INTERFACE I_ChainController

METHOD addChain : I_ChainController 
VAR_INPUT
	itfChain : I_Chain;
END_VAR
END_METHOD

METHOD releaseForChain : I_ChainController
VAR_INPUT
	sChainToRelease : STRING;
	itfCommissioner : I_Chain;
END_VAR
END_METHOD

METHOD releaseFromChain : I_ChainController
VAR_INPUT
	sChainReleasing : STRING;
	itfContractor : I_Chain;
END_VAR
END_METHOD

METHOD releaseResult : Bool
VAR_INPUT
	itfRequester : I_Chain;
END_VAR
END_METHOD

END_INTERFACE

(* stored: Version 1.1.0.1, ProductVersion 3.1.4024.0
   Itf I_ChainController: Id {e3242905-8342-45d0-836e-b3cfbaafbabd}
   Method addChain: Id {701c894c-d937-4641-9a3f-44dfc24f176f}
   Method releaseForChain: Id {4bbaaa44-534a-41a1-80a4-5024df2c342e}
   Method releaseFromChain: Id {30f3d0cf-7fcb-4b64-bfe5-7dabfd1a983d}
   Method releaseResult: Id {e1fbf38c-e6a7-4739-ba2e-e2a5ca4593b6} *)
